FUNCTION_BLOCK SM_LineRegulator EXTENDS StateMachine
VAR_INPUT
END_VAR
VAR_OUTPUT
END_VAR
VAR
	fbTurntable : Turntable;
	aRollerConveyors : ARRAY[1..3] OF RollerConveyor;
END_VAR

Super^();

METHOD PROTECTED   Busy : BOOL
VAR_INPUT
END_VAR
END_METHOD

METHOD PROTECTED  Error : BOOL
VAR_INPUT
END_VAR
END_METHOD

METHOD PROTECTED  Idle : BOOL
VAR_INPUT
END_VAR
END_METHOD

METHOD PROTECTED  Init : BOOL
VAR_INPUT
END_VAR
Start();
END_METHOD

METHOD PROTECTED  Prepare : BOOL
VAR_INPUT
END_VAR
END_METHOD

METHOD PROTECTED  Ready : BOOL
VAR_INPUT
END_VAR
END_METHOD

METHOD PROTECTED  Waiting : BOOL
VAR_INPUT
END_VAR
END_METHOD

END_FUNCTION_BLOCK

(* stored: Version 1.1.0.1, ProductVersion 3.1.4024.0
   POU SM_LineRegulator: Id {ca3d4937-9986-4e8e-b7ee-5deb908a267b}, SpecialFunc None
   Method Busy: Id {5f49f79a-dd7d-411c-abbd-7df000596daa}
   Method Error: Id {239c3776-b310-4e44-8c9a-3b822be85443}
   Method Idle: Id {8991d786-6df6-47cb-9e47-3ad5344b1f79}
   Method Init: Id {61709bba-0e18-44c6-961b-6552433808b6}
   Method Prepare: Id {6b592004-8cf2-4348-b3e7-517e0f77b060}
   Method Ready: Id {f9a8f055-f81d-4c23-82e5-c30d5480dd80}
   Method Waiting: Id {d736384e-810f-4ff5-9820-b539fdf97b0f} *)
